(* Logix 5000 project; controller AMP_Servo_Demo vendor 1 type 14 code 154 rev 32.15; software revision 32.05; part 4 of 5 *)

ADD_ON_INSTRUCTION AMP_Relative_Move   (* revision 1.0, vendor Applied Motion Products Inc. *)
// Applied Motion - Motor Relative Move - AOI
// Help:
// The Relative Move AOI is used to move an axis by a specified distance (positive or negative) relative to its currently commanded position(FL).
VAR_IN_OUT
   Input : DINT[20]; {required}   // Drive Input Assembly
        [12]   // Digital_Outputs
        [7]   // Drive_Temperature
        [2]   // Control_Mode
        [3]   // Status_Code
        [9]   // Second_Encoder_Position
        [16]   // Analog_Input1
        [17]   // Analog_Input2
        [4]   // Alarm_Code
        [18]   // Torque_Limit
        [5]   // Supply_Voltage
        [6]   // Applied_Torque
        [10]   // Position_Error
        [13]   // Digital_Inputs
        [14]   // Analog_Output1
        [15]   // Analog_Output2
        [1]   // OpCode1_Received
        [8]   // Encoder_Position
        [0]   // Control_Word_Received
        [11]   // Actual_Velocity_RPS
        [19]   // Second_Encoder_Speed
   Output : DINT[11]; {required}   // Drive Output Assembly
        [0]   // Control Word
        [5]   // Porifle Acceleration
        [6]   // Profile Deceleration
        [7]   // Target Torque
        [4]   // Target Velocity
        [10]   // Reserved
        [3]   // Target Pos
        [1]   // OpCode 1
        [2]   // OpCode 2
        [8]   // OpCode 3
        [9]   // OpCode 4
END_VAR
VAR_INPUT
   Start : BOOL; {required}   // Start the Relative Move
   Distance : DINT; {required}   // Relative Distance to Move (negative = reverse)
   Speed_rps : REAL; {required}   // Velocity of Move (rev/sec)
   Acc : REAL; {required}   // Acceleration of Move (rev/s/s)
   Dec : REAL; {required}   // Deceleration of Move (rev/s/s)
END_VAR
VAR_OUTPUT
   Sent : BOOL; {access Read Only, visible}   // Move has been sent to drive
   In_Progress : BOOL; {access Read Only, visible}   // Move in progress
   Done : BOOL; {access Read Only, visible}   // Move completed without errors - desired position reached
   Error : BOOL; {access Read Only, visible}   // Move failed to complete - drive not ready or faulted
   State : DINT := 10; {access Read Only}   // Internal state of progress
END_VAR
VAR
   Loc_StatusCode : AMP_Status_Word_Servo; {access None}
   Loc_Rel_ONS : BOOL;
   Loc_Input_Assembly : AMP_Input_Assembly_Servo_v2; {access None}
   Loc_Command_Timeout : TIMER := (PRE := 2000); {access None}   // Timer to output fault if command is not Done
END_VAR

ROUTINE Logic   (* ladder *)
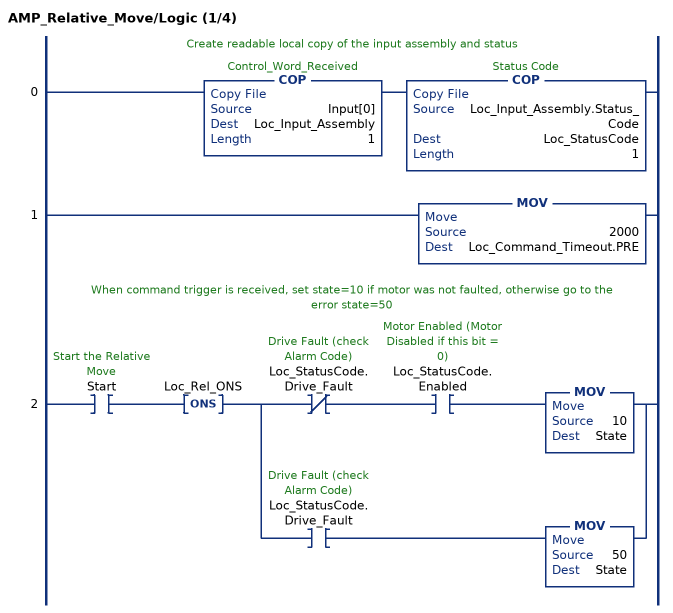
   // Create readable local copy of the input assembly and status
   0: COP(Input[0],Loc_Input_Assembly,1)COP(Loc_Input_Assembly.Status_Code,Loc_StatusCode,1);
   1: MOV(2000,Loc_Command_Timeout.PRE);
   // When command trigger is received, set state=10 if motor was not faulted, otherwise go to the error state=50
   2: XIC(Start)ONS(Loc_Rel_ONS)[XIO(Loc_StatusCode.Drive_Fault) XIC(Loc_StatusCode.Enabled) MOV(10,State) ,XIC(Loc_StatusCode.Drive_Fault) MOV(50,State) ];
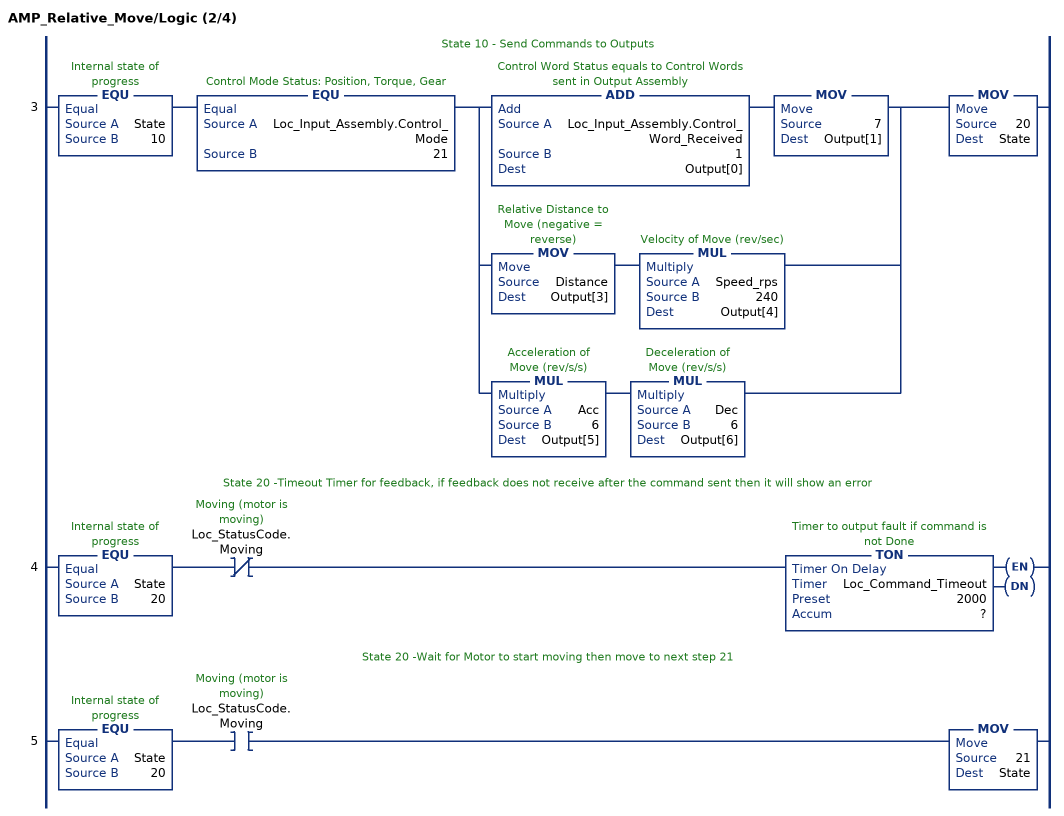
   // State 10 - Send Commands to Outputs
   3: EQU(State,10)EQU(Loc_Input_Assembly.Control_Mode,21)[ADD(Loc_Input_Assembly.Control_Word_Received,1,Output[0]) MOV(7,Output[1]) ,MOV(Distance,Output[3]) MUL(Speed_rps,240,Output[4]) ,MUL(Acc,6,Output[5]) MUL(Dec,6,Output[6]) ]MOV(20,State);
   // State 20 -Timeout Timer for feedback, if feedback does not receive after the command sent then it will show an error
   4: EQU(State,20)XIO(Loc_StatusCode.Moving)TON(Loc_Command_Timeout,?,?);
   // State 20 -Wait for Motor to start moving then move to next step 21
   5: EQU(State,20)XIC(Loc_StatusCode.Moving)MOV(21,State);
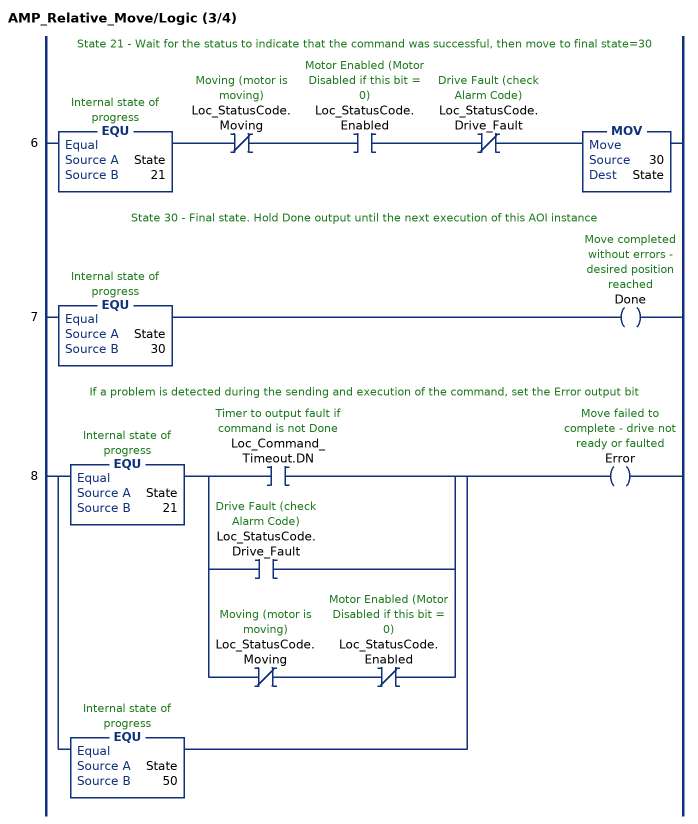
   // State 21 - Wait for the status to indicate that the command was successful, then move to final state=30
   6: EQU(State,21)XIO(Loc_StatusCode.Moving)XIC(Loc_StatusCode.Enabled)XIO(Loc_StatusCode.Drive_Fault)MOV(30,State);
   // State 30 - Final state. Hold Done output until the next execution of this AOI instance
   7: EQU(State,30)OTE(Done);
   // If a problem is detected during the sending and execution of the command, set the Error output bit
   8: [EQU(State,21) [XIC(Loc_Command_Timeout.DN) ,XIC(Loc_StatusCode.Drive_Fault) ,XIO(Loc_StatusCode.Moving) XIO(Loc_StatusCode.Enabled) ] ,EQU(State,50) ]OTE(Error);
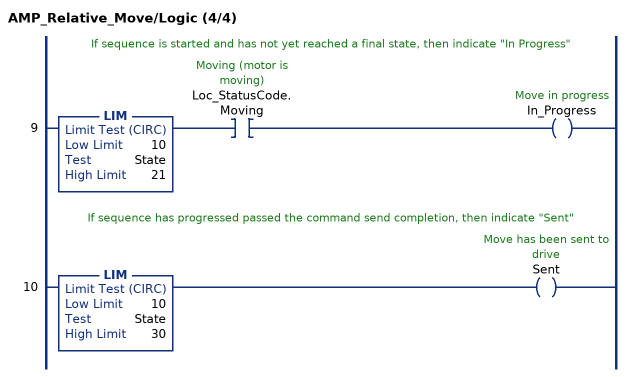
   // If sequence is started and has not yet reached a final state, then indicate "In Progress"
   9: LIM(10,State,21)XIC(Loc_StatusCode.Moving)OTE(In_Progress);
   // If sequence has progressed passed the command send completion, then indicate "Sent"
   10: LIM(10,State,30)OTE(Sent);
END_ROUTINE
END_ADD_ON_INSTRUCTION

ADD_ON_INSTRUCTION AMP_SCL_Command   (* revision 1.0, vendor Applied Motion Products Inc. *)
// Applied Motion - Motor SCL Command - AOI
// Help:
// The SCL Command Execute AOI executes selected SCL commands (as listed under “Available SCL Commands” in the reference manual).
VAR_IN_OUT
   Input : DINT[20]; {required}   // Drive Input Assembly
        [12]   // Digital_Outputs
        [7]   // Drive_Temperature
        [2]   // Control_Mode
        [9]   // Second_Encoder_Position
        [3]   // Status_Code
        [16]   // Analog_Input1
        [17]   // Analog_Input2
        [18]   // Torque_Limit
        [4]   // Alarm_Code
        [5]   // Supply_Voltage
        [6]   // Applied_Torque
        [10]   // Position_Error
        [13]   // Digital_Inputs
        [14]   // Analog_Output1
        [15]   // Analog_Output2
        [1]   // OpCode1_Received
        [8]   // Encoder_Position
        [0]   // Control_Word_Received
        [11]   // Actual_Velocity_RPS
        [19]   // Second_Encoder_Speed
   Output : DINT[11]; {required}   // Drive Output Assembly
        [0]   // Control Word
        [5]   // Porifle Acceleration
        [6]   // Profile Deceleration
        [7]   // Target Torque
        [4]   // Target Velocity
        [10]   // Reserved
        [3]   // Target Pos
        [1]   // OpCode 1
        [2]   // OpCode 2
        [8]   // OpCode 3
        [9]   // OpCode 4
END_VAR
VAR_INPUT
   Execute : BOOL; {required}   // Execute the SCL command
   SCL_Command : INT; {required}   // SCL Command Characters (always 2)
   Reg1 : DINT; {required}   // Data / SCL Register 1
   Reg2 : DINT; {required}   // Data / SCL Register 2
END_VAR
VAR_OUTPUT
   Sent : BOOL; {access Read Only, visible}   // Command has been sent to drive
   In_Progress : BOOL; {access Read Only, visible}   // Command in progress
   Done : BOOL; {access Read Only, visible}   // Command completed without errors
   Error : BOOL; {access Read Only, visible}   // Command failed
   State : DINT := 10; {access Read Only}   // Internal state of progress
END_VAR
VAR
   Loc_StatusCode : AMP_Status_Word_Servo; {access None}
   Loc_SCL_ONS : BOOL;
   Loc_Input_Assembly : AMP_Input_Assembly_Servo_v2; {access None}
END_VAR

ROUTINE Logic   (* ladder *)
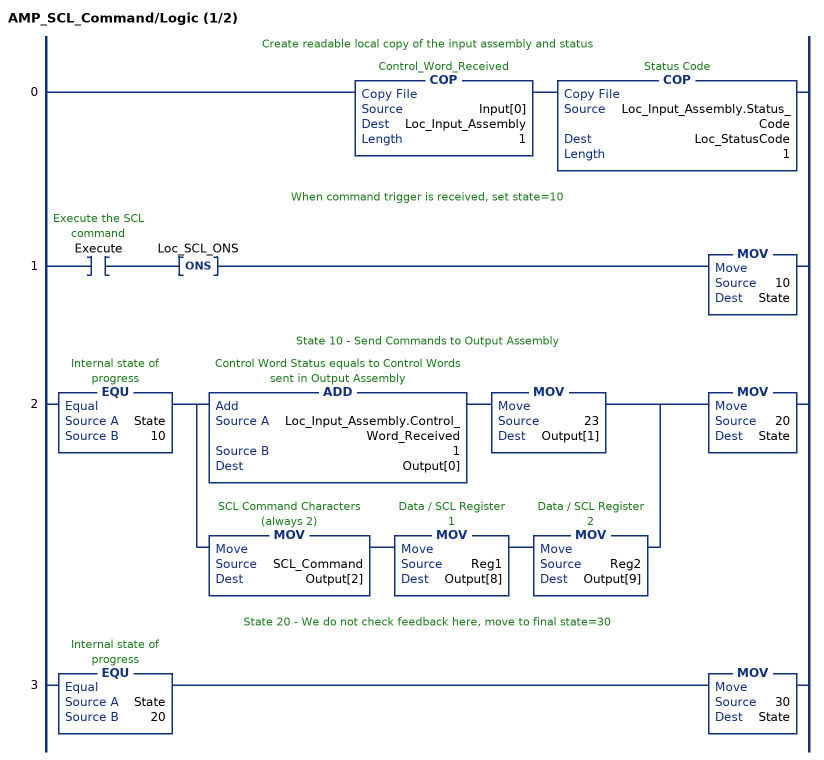
   // Create readable local copy of the input assembly and status
   0: COP(Input[0],Loc_Input_Assembly,1)COP(Loc_Input_Assembly.Status_Code,Loc_StatusCode,1);
   // When command trigger is received, set state=10
   1: XIC(Execute)ONS(Loc_SCL_ONS)MOV(10,State);
   // State 10 - Send Commands to Output Assembly
   2: EQU(State,10)[ADD(Loc_Input_Assembly.Control_Word_Received,1,Output[0]) MOV(23,Output[1]) ,MOV(SCL_Command,Output[2]) MOV(Reg1,Output[8]) MOV(Reg2,Output[9]) ]MOV(20,State);
   // State 20 - We do not check feedback here, move to final state=30
   3: EQU(State,20)MOV(30,State);
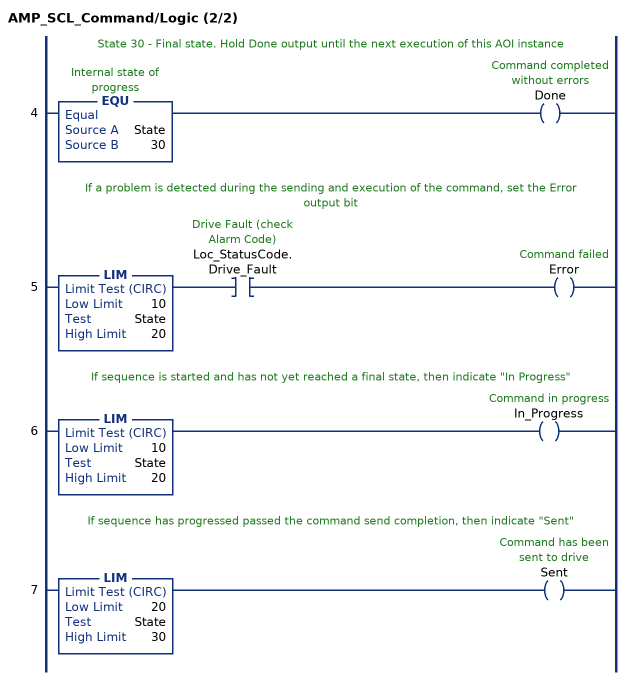
   // State 30 - Final state. Hold Done output until the next execution of this AOI instance
   4: EQU(State,30)OTE(Done);
   // If a problem is detected during the sending and execution of the command, set the Error output bit
   5: LIM(10,State,20)XIC(Loc_StatusCode.Drive_Fault)OTE(Error);
   // If sequence is started and has not yet reached a final state, then indicate "In Progress"
   6: LIM(10,State,20)OTE(In_Progress);
   // If sequence has progressed passed the command send completion, then indicate "Sent"
   7: LIM(20,State,30)OTE(Sent);
END_ROUTINE
END_ADD_ON_INSTRUCTION

ADD_ON_INSTRUCTION AMP_Set_Position   (* revision 1.0 *)
// Applied Motion - Motor Set Position - AOI
// Help:
// The Motor Enable AOI restores drive current to motor.
VAR_IN_OUT
   Input : DINT[20]; {required}   // Drive Input Assembly
        [12]   // Digital_Outputs
        [7]   // Drive_Temperature
        [2]   // Control_Mode
        [3]   // Status_Code
        [9]   // Second_Encoder_Position
        [16]   // Analog_Input1
        [17]   // Analog_Input2
        [4]   // Alarm_Code
        [18]   // Torque_Limit
        [5]   // Supply_Voltage
        [6]   // Applied_Torque
        [10]   // Position_Error
        [13]   // Digital_Inputs
        [14]   // Analog_Output1
        [15]   // Analog_Output2
        [1]   // OpCode1_Received
        [0]   // Control_Word_Received
        [11]   // Actual_Velocity_RPS
        [8]   // Encoder_Position
        [19]   // Second_Encoder_Speed
   Output : DINT[11]; {required}   // Drive Output Assembly
        [0]   // Control Word
        [5]   // Porifle Acceleration
        [6]   // Profile Deceleration
        [7]   // Target Torque
        [4]   // Target Velocity
        [10]   // Reserved
        [3]   // Target Pos
        [1]   // OpCode 1
        [2]   // OpCode 2
        [8]   // OpCode 3
        [9]   // OpCode 4
END_VAR
VAR_INPUT
   Execute : BOOL; {required}   // Execute the SCL command EP
   Position : DINT; {required}   // Position SetPoint DINT value
END_VAR
VAR_OUTPUT
   Sent : BOOL; {access Read Only, visible}   // Command has been sent to drive
   In_Progress : BOOL; {access Read Only, visible}   // Command in progress
   Done : BOOL; {access Read Only, visible}   // Command completed without errors - Drive is Homed
   Error : BOOL; {access Read Only, visible}   // Command failed
   State : DINT := 10; {access Read Only}   // Internal state of progress
END_VAR
VAR
   Loc_StatusCode : AMP_Status_Word_Servo;
   Loc_Input_Assembly : AMP_Input_Assembly_Servo_v2;
   Loc_SCL_ONS : BOOL;
   Loc_Reg2 : DINT;   // Data / SCL Register 2
   Loc_Reg1 : DINT;   // Data / SCL Register 1
   Loc_SCL_Command : INT := 'EP';   // SCL Command Characters (always 2)
END_VAR

ROUTINE Logic   (* ladder *)
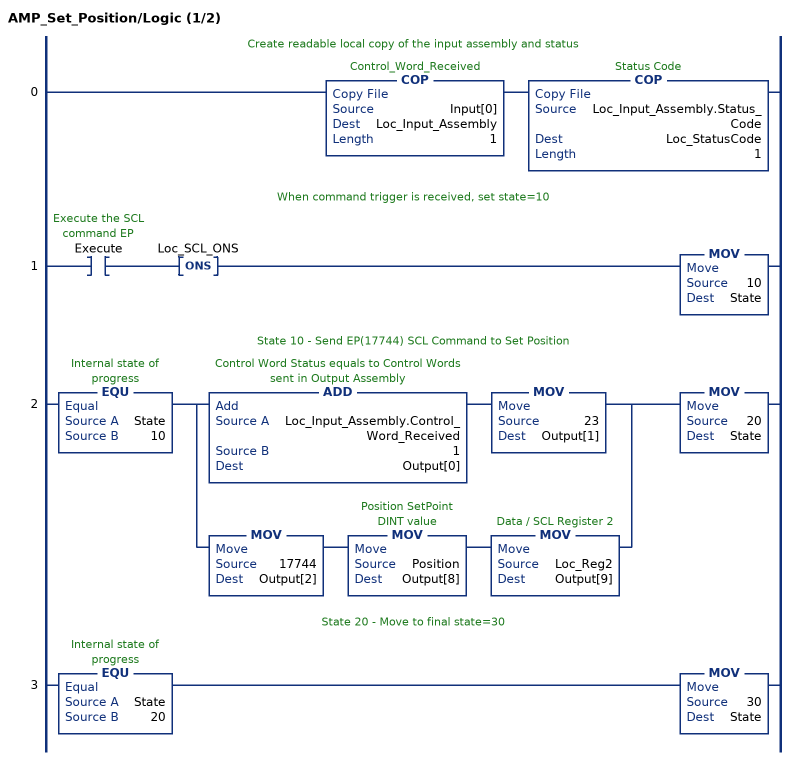
   // Create readable local copy of the input assembly and status
   0: COP(Input[0],Loc_Input_Assembly,1)COP(Loc_Input_Assembly.Status_Code,Loc_StatusCode,1);
   // When command trigger is received, set state=10
   1: XIC(Execute)ONS(Loc_SCL_ONS)MOV(10,State);
   // State 10 - Send EP(17744) SCL Command to Set Position
   2: EQU(State,10)[ADD(Loc_Input_Assembly.Control_Word_Received,1,Output[0]) MOV(23,Output[1]) ,MOV(17744,Output[2]) MOV(Position,Output[8]) MOV(Loc_Reg2,Output[9]) ]MOV(20,State);
   // State 20 - Move to final state=30
   3: EQU(State,20)MOV(30,State);
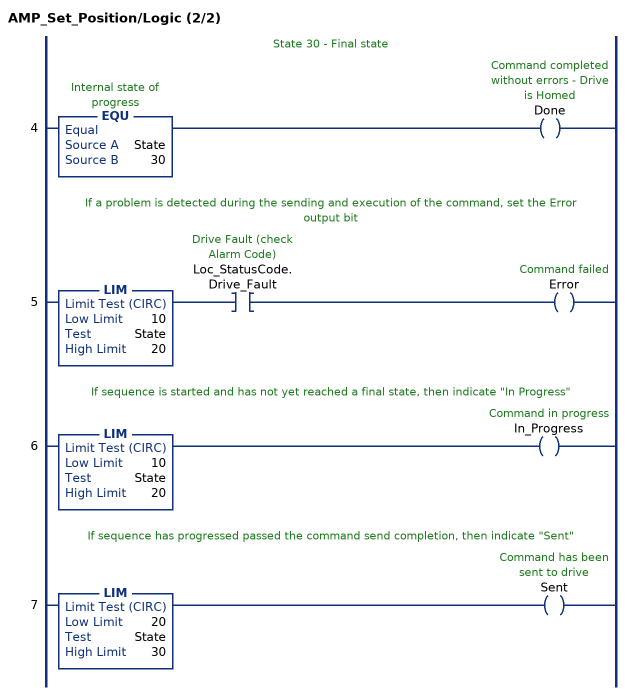
   // State 30 - Final state
   4: EQU(State,30)OTE(Done);
   // If a problem is detected during the sending and execution of the command, set the Error output bit
   5: LIM(10,State,20)XIC(Loc_StatusCode.Drive_Fault)OTE(Error);
   // If sequence is started and has not yet reached a final state, then indicate "In Progress"
   6: LIM(10,State,20)OTE(In_Progress);
   // If sequence has progressed passed the command send completion, then indicate "Sent"
   7: LIM(20,State,30)OTE(Sent);
END_ROUTINE
END_ADD_ON_INSTRUCTION

ADD_ON_INSTRUCTION AMP_Status_Code   (* revision 1.0, vendor Applied Motion Products Inc. *)
// Applied Motion - Status Code(SC) AOI
// Help:
// The Status Code AOI uses the raw data stored in the Status Code word (Element 0 from Input Assembly) to set individual appropriately named boolean outputs.
VAR_INPUT
   Input : DINT; {required}   // Element 4 from Drive Input Assembly
END_VAR
VAR_OUTPUT
   Motor_Enabled : BOOL; {access Read Only, visible}   // Motor is Enabled(Brake is released if applicable)
   Sampling : BOOL; {access Read Only, visible}   // Sampling (Luna software oscilloscope function opens)
   Drive_Fault : BOOL; {access Read Only, visible}   // Drive has fault, Motor Disabled
   In_Position : BOOL; {access Read Only, visible}   // Motor is in Position, it is standstill
   Moving : BOOL; {access Read Only, visible}   // Motor is Moving
   Jogging : BOOL; {access Read Only, visible}   // Motor is Jogging
   Stopping : BOOL; {access Read Only, visible}   // Motor is Stopping (Decelerating)
   Waiting : BOOL; {access Read Only, visible}   // Wait for Input Signal (e.g. follow WI command)
   Saving : BOOL; {access Read Only, visible}   // Drive is Saving Parameters
   Alarm_Present : BOOL; {access Read Only, visible}   // Dirve has alram present, fault and warning
   Homing : BOOL; {access Read Only, visible}   // Motor is Homing
   Wait_Time : BOOL; {access Read Only, visible}   // Waiting for an input (executing WD or WT command/delay after homing)
   Wizard_Running : BOOL; {access Read Only, visible}   // Wizard Running, Drive internal status
   Checking_Encoder : BOOL; {access Read Only, visible}   // Drive is checking encoder, Drive internal status
   Q_Program_Running : BOOL; {access Read Only, visible}   // Q Program is executing
   Servo_Ready : BOOL; {access Read Only, visible}   // Servo is ready
   CSP_Following : BOOL; {access Read Only, visible}   // CSP following internal status
   In_Velocity : BOOL; {access Read Only, visible}   // Motor is in Velocity
   Zero_Speed : BOOL; {access Read Only, visible}   // Motor is not moving
   Torque_Reached : BOOL; {access Read Only, visible}   // Torque Arrival
   In_Torque : BOOL; {access Read Only, visible}   // Consistent Torque
   Group2_PID : BOOL; {access Read Only, visible}   // The second set of gain is in operation
   Secondary_Control_Mode : BOOL; {access Read Only, visible}   // The second control mode is in operation
   Velocity_Reached : BOOL; {access Read Only, visible}   // Velocity is reached
   Homing_Complete : BOOL; {access Read Only, visible}   // Homing has been completed
END_VAR

ROUTINE Logic   (* ladder *)
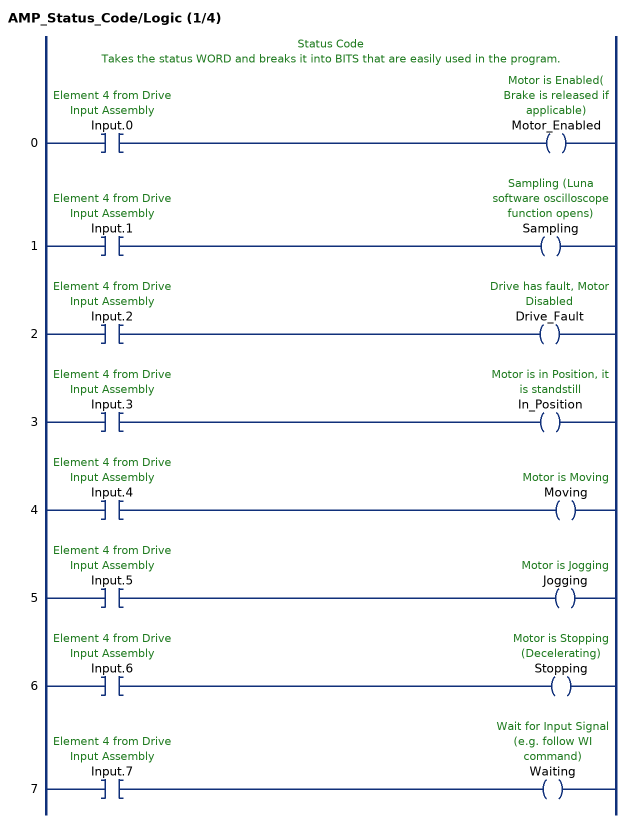
   // Status Code
   // Takes the status WORD and breaks it into BITS that are easily used in the program.
   0: XIC(Input.0)OTE(Motor_Enabled);
   1: XIC(Input.1)OTE(Sampling);
   2: XIC(Input.2)OTE(Drive_Fault);
   3: XIC(Input.3)OTE(In_Position);
   4: XIC(Input.4)OTE(Moving);
   5: XIC(Input.5)OTE(Jogging);
   6: XIC(Input.6)OTE(Stopping);
   7: XIC(Input.7)OTE(Waiting);
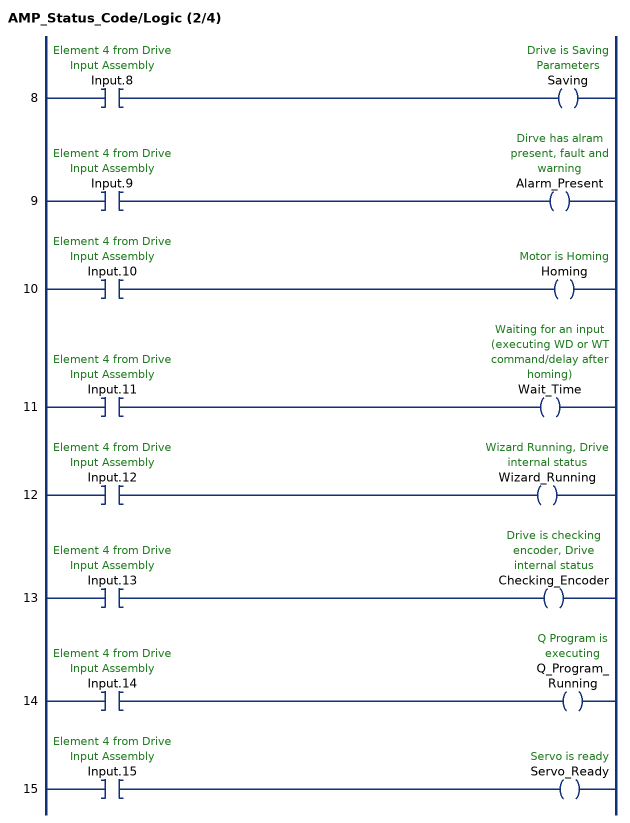
   8: XIC(Input.8)OTE(Saving);
   9: XIC(Input.9)OTE(Alarm_Present);
   10: XIC(Input.10)OTE(Homing);
   11: XIC(Input.11)OTE(Wait_Time);
   12: XIC(Input.12)OTE(Wizard_Running);
   13: XIC(Input.13)OTE(Checking_Encoder);
   14: XIC(Input.14)OTE(Q_Program_Running);
   15: XIC(Input.15)OTE(Servo_Ready);
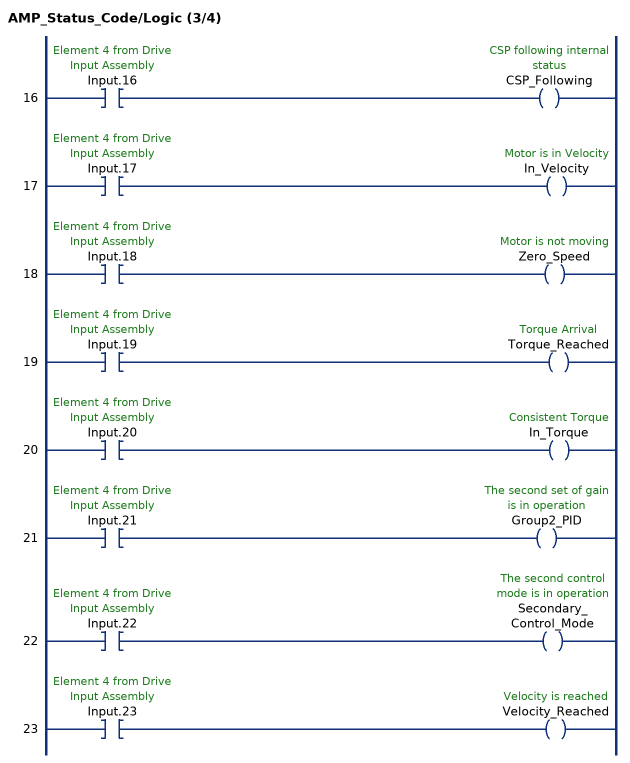
   16: XIC(Input.16)OTE(CSP_Following);
   17: XIC(Input.17)OTE(In_Velocity);
   18: XIC(Input.18)OTE(Zero_Speed);
   19: XIC(Input.19)OTE(Torque_Reached);
   20: XIC(Input.20)OTE(In_Torque);
   21: XIC(Input.21)OTE(Group2_PID);
   22: XIC(Input.22)OTE(Secondary_Control_Mode);
   23: XIC(Input.23)OTE(Velocity_Reached);
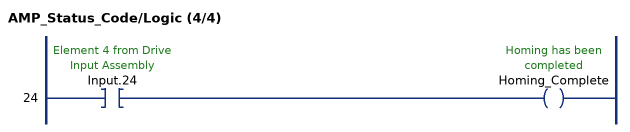
   24: XIC(Input.24)OTE(Homing_Complete);
END_ROUTINE
END_ADD_ON_INSTRUCTION

ADD_ON_INSTRUCTION AMP_Torque_Control   (* revision 1.0 *)
// Applied Motion - Motor Torque - AOI
// Use Normal/Crash Stop AOI to Stop Torque
// Help:
// The AOI switch Control mode to Torque mode and apply Torque. Use Normal stop or Crash stop AOI to stop applying torque.
// Target Torque Percentage is Limit by Torque Limit shown in Input Assembly.
VAR_IN_OUT
   Input : DINT[20]; {required}   // Drive Input Assembly
        [12]   // Digital_Outputs
        [7]   // Drive_Temperature
        [2]   // Control_Mode
        [3]   // Status_Code
        [16]   // Analog_Input1
        [17]   // Analog_Input2
        [9]   // Second_Encoder_Position
        [4]   // Alarm_Code
        [18]   // Torque_Limit
        [5]   // Supply_Voltage
        [6]   // Applied_Torque
        [0]   // Control_Word_Received
        [11]   // Actual_Velocity_RPS
        [19]   // Second_Encoder_Speed
        [10]   // Position_Error
        [13]   // Digital_Inputs
        [14]   // Analog_Output1
        [15]   // Analog_Output2
        [1]   // OpCode1_Received
        [8]   // Encoder_Position
   Output : DINT[11]; {required}   // Drive Output Assembly
        [0]   // Control Word
        [5]   // Porifle Acceleration
        [6]   // Profile Deceleration
        [7]   // Target Torque
        [4]   // Target Velocity
        [10]   // Reserved
        [3]   // Target Pos
        [1]   // OpCode 1
        [2]   // OpCode 2
        [8]   // OpCode 3
        [9]   // OpCode 4
END_VAR
VAR_INPUT
   Start : BOOL; {required}   // Start Applying Torque (on rising edge)
   Target_Torque_Percentage : INT := 10; {required}   // Target Torque Percentage, for reverse direction use Negative value
   Torque_Ramp : INT; {required}   // Torque Ramp (0.1%/sec)
   Speed_Limit_rps : REAL; {required}   // Torque Speed Limit in rps
   Acc : REAL; {required}   // Acceleration rev/s/s
   Dec : REAL; {required}   // Deceleration rev/s/s
END_VAR
VAR_OUTPUT
   Sent : BOOL; {access Read Only, visible}   // Command has been sent to drive
   In_Progress : BOOL; {access Read Only, visible}   // Command is in progress
   Done : BOOL; {access Read Only, visible}   // Command completed without errors
   Error : BOOL; {access Read Only, visible}   // Command Failed
   State : DINT := 10; {access Read Only}   // Internal state of progress
END_VAR
VAR
   Loc_StatusCode : AMP_Status_Word_Servo;
   Loc_Input_Assembly : AMP_Input_Assembly_Servo_v2;
   Loc_Torque_ONS : BOOL;
   Loc_Command_Wait : TIMER := (PRE := 100); {access None}   // Wait Timer for New Command
END_VAR

ROUTINE Logic   (* ladder *)
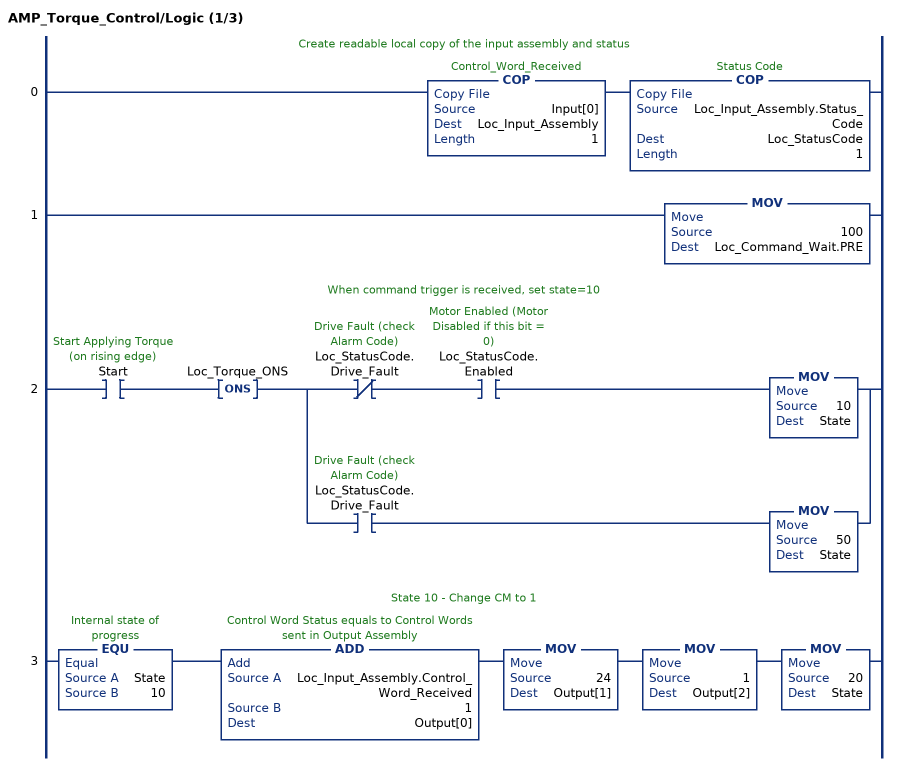
   // Create readable local copy of the input assembly and status
   0: COP(Input[0],Loc_Input_Assembly,1)COP(Loc_Input_Assembly.Status_Code,Loc_StatusCode,1);
   1: MOV(100,Loc_Command_Wait.PRE);
   // When command trigger is received, set state=10
   2: XIC(Start)ONS(Loc_Torque_ONS)[XIO(Loc_StatusCode.Drive_Fault) XIC(Loc_StatusCode.Enabled) MOV(10,State) ,XIC(Loc_StatusCode.Drive_Fault) MOV(50,State) ];
   // State 10 - Change CM to 1
   3: EQU(State,10)ADD(Loc_Input_Assembly.Control_Word_Received,1,Output[0])MOV(24,Output[1])MOV(1,Output[2])MOV(20,State);
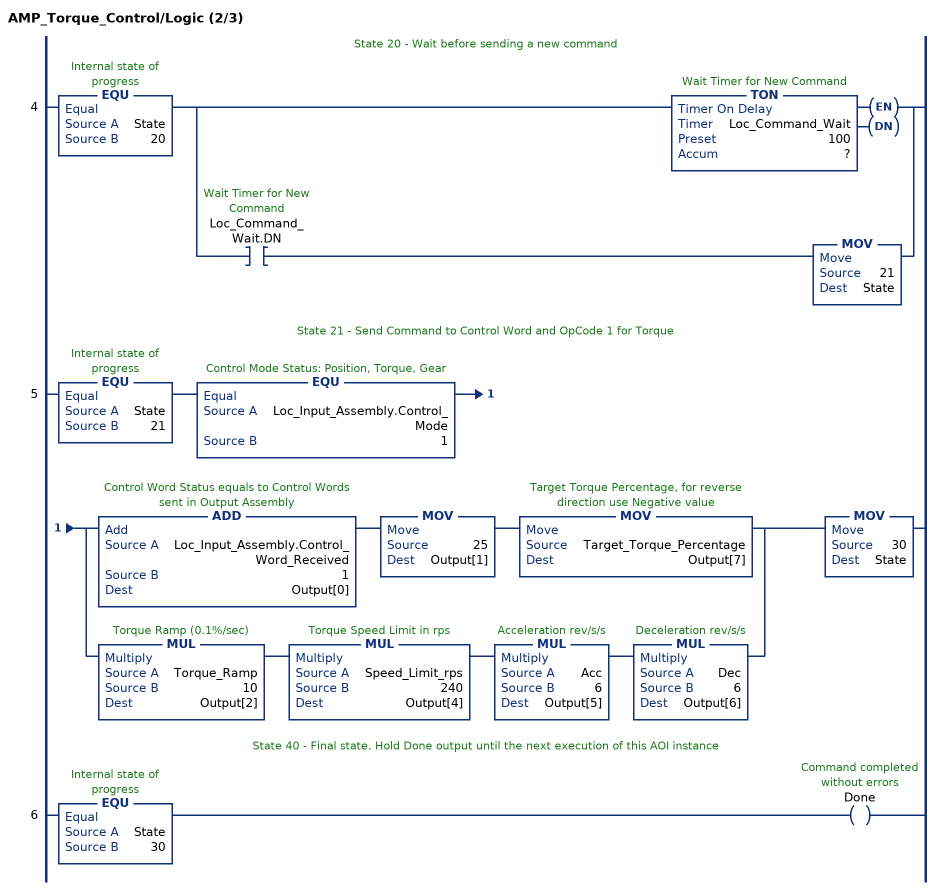
   // State 20 - Wait before sending a new command
   4: EQU(State,20)[TON(Loc_Command_Wait,?,?) ,XIC(Loc_Command_Wait.DN) MOV(21,State) ];
   // State 21 - Send Command to Control Word and OpCode 1 for Torque
   5: EQU(State,21)EQU(Loc_Input_Assembly.Control_Mode,1)[ADD(Loc_Input_Assembly.Control_Word_Received,1,Output[0]) MOV(25,Output[1]) MOV(Target_Torque_Percentage,Output[7]) ,MUL(Torque_Ramp,10,Output[2]) MUL(Speed_Limit_rps,240,Output[4]) MUL(Acc,6,Output[5]) MUL(Dec,6,Output[6]) ]MOV(30,State);
   // State 40 - Final state. Hold Done output until the next execution of this AOI instance
   6: EQU(State,30)OTE(Done);
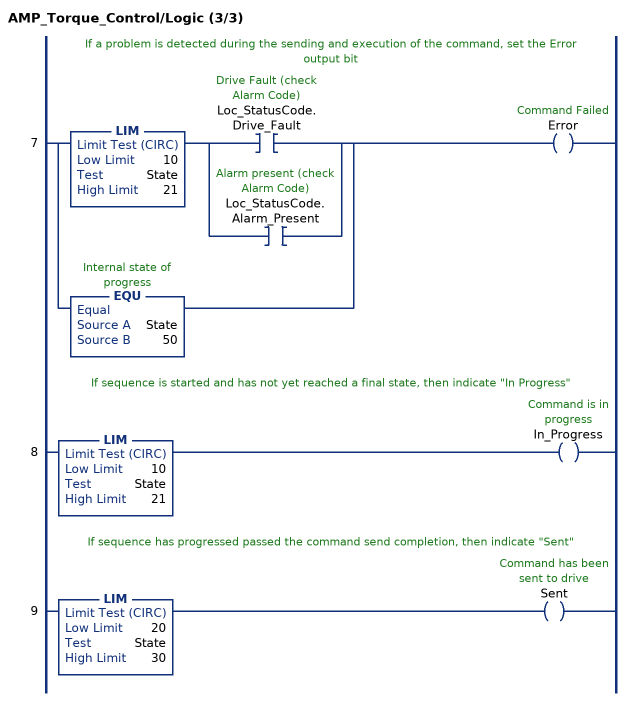
   // If a problem is detected during the sending and execution of the command, set the Error output bit
   7: [LIM(10,State,21) [XIC(Loc_StatusCode.Drive_Fault) ,XIC(Loc_StatusCode.Alarm_Present) ] ,EQU(State,50) ]OTE(Error);
   // If sequence is started and has not yet reached a final state, then indicate "In Progress"
   8: LIM(10,State,21)OTE(In_Progress);
   // If sequence has progressed passed the command send completion, then indicate "Sent"
   9: LIM(20,State,30)OTE(Sent);
END_ROUTINE
END_ADD_ON_INSTRUCTION

ADD_ON_INSTRUCTION AMP_Update_Jog_Speed   (* revision 1.0 *)
// Applied Motion - Motor Update Speed for Jog Only- AOI
// Help:
// This AOI updates the Jogging Speed either in Positive or Negative direction(CS). User need to use Normal Stop or Crash Stop AOI to Stop Jogging.
VAR_IN_OUT
   Input : DINT[20]; {required}   // Drive Input Assembly
        [12]   // Digital_Outputs
        [7]   // Drive_Temperature
        [2]   // Control_Mode
        [3]   // Status_Code
        [9]   // Second_Encoder_Position
        [16]   // Analog_Input1
        [17]   // Analog_Input2
        [4]   // Alarm_Code
        [19]   // Second_Encoder_Speed
        [18]   // Torque_Limit
        [5]   // Supply_Voltage
        [0]   // Control_Word_Received
        [6]   // Applied_Torque
        [11]   // Actual_Velocity_RPS
        [10]   // Position_Error
        [13]   // Digital_Inputs
        [14]   // Analog_Output1
        [15]   // Analog_Output2
        [1]   // OpCode1_Received
        [8]   // Encoder_Position
   Output : DINT[11]; {required}   // Drive Output Assembly
        [4]   // Jog Speed (0.25 rev/min)
        [0]   // Control Word
        [5]   // Porifle Acceleration
        [6]   // Profile Deceleration
        [7]   // Target Torque
        [10]   // Reserved
        [3]   // Target Pos
        [1]   // OpCode 1
        [2]   // OpCode 2
        [8]   // OpCode 3
        [9]   // OpCode 4
END_VAR
VAR_INPUT
   Update : BOOL; {required}   // Update Speed Command
   Speed_rps : REAL; {required}   // Velocity of Jog (rev/sec)(negative=reverse)
END_VAR
VAR_OUTPUT
   Sent : BOOL; {access Read Only, visible}   // Update Speed Command has been sent to drive
   In_Progress : BOOL; {access Read Only, visible}   // Update Speed Command in progress
   Done : BOOL; {access Read Only, visible}   // Update Speed command completed without errors
   Error : BOOL; {access Read Only, visible}   // Command failed
   State : DINT := 10; {access Read Only}   // Internal state of progress
END_VAR
VAR
   Loc_StatusCode : AMP_Status_Word_Servo;
   Command_Timeout : TIMER := (PRE := 2000);   // Timer to make sure command value was 0 before sending a new command
   Loc_Input_Assembly : AMP_Input_Assembly_Servo_v2;
   Loc_Jog_ONS : BOOL;
   Command_Reset : TIMER; {access None}   // Timer to make sure command value was 0 before sending a new command
END_VAR

ROUTINE Logic   (* ladder *)
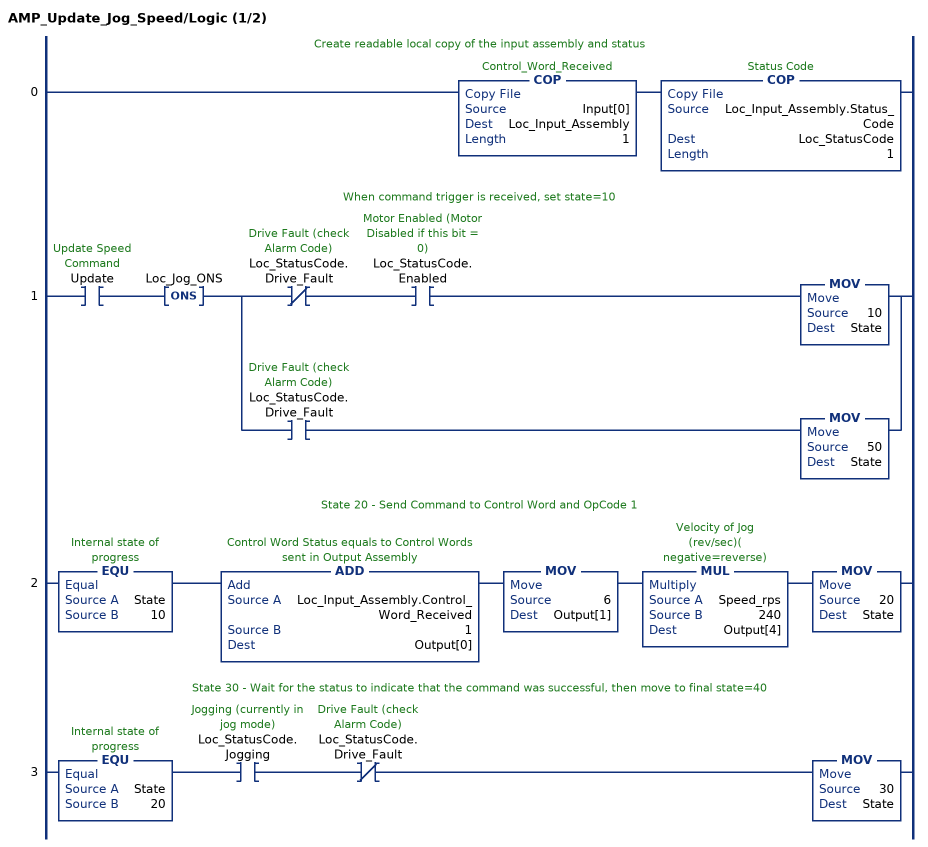
   // Create readable local copy of the input assembly and status
   0: COP(Input[0],Loc_Input_Assembly,1)COP(Loc_Input_Assembly.Status_Code,Loc_StatusCode,1);
   // When command trigger is received, set state=10
   1: XIC(Update)ONS(Loc_Jog_ONS)[XIO(Loc_StatusCode.Drive_Fault) XIC(Loc_StatusCode.Enabled) MOV(10,State) ,XIC(Loc_StatusCode.Drive_Fault) MOV(50,State) ];
   // State 20 - Send Command to Control Word and OpCode 1
   2: EQU(State,10)ADD(Loc_Input_Assembly.Control_Word_Received,1,Output[0])MOV(6,Output[1])MUL(Speed_rps,240,Output[4])MOV(20,State);
   // State 30 - Wait for the status to indicate that the command was successful, then move to final state=40
   3: EQU(State,20)XIC(Loc_StatusCode.Jogging)XIO(Loc_StatusCode.Drive_Fault)MOV(30,State);
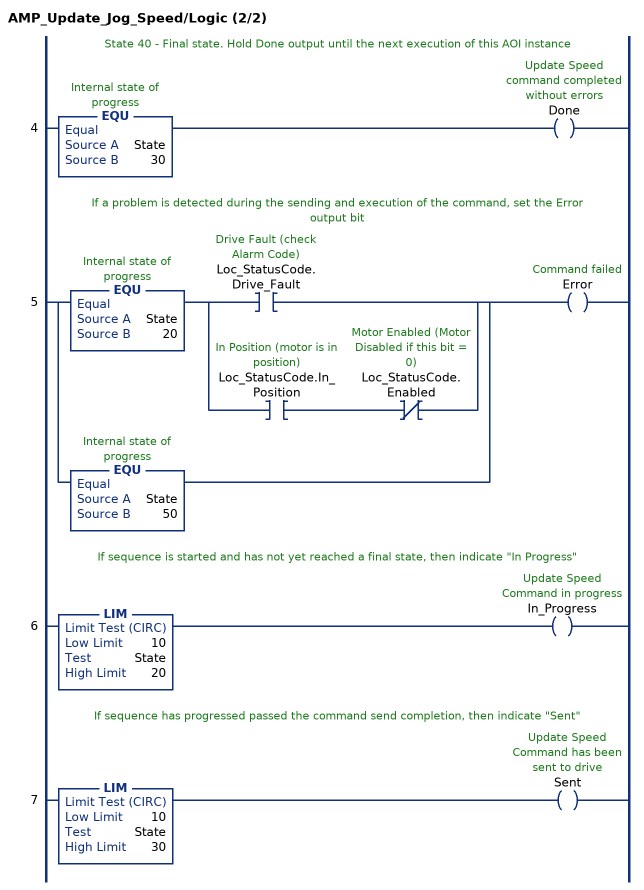
   // State 40 - Final state. Hold Done output until the next execution of this AOI instance
   4: EQU(State,30)OTE(Done);
   // If a problem is detected during the sending and execution of the command, set the Error output bit
   5: [EQU(State,20) [XIC(Loc_StatusCode.Drive_Fault) ,XIC(Loc_StatusCode.In_Position) XIO(Loc_StatusCode.Enabled) ] ,EQU(State,50) ]OTE(Error);
   // If sequence is started and has not yet reached a final state, then indicate "In Progress"
   6: LIM(10,State,20)OTE(In_Progress);
   // If sequence has progressed passed the command send completion, then indicate "Sent"
   7: LIM(10,State,30)OTE(Sent);
END_ROUTINE
END_ADD_ON_INSTRUCTION

VAR_GLOBAL   (* controller tags *)
   Amp_01_MSG1 : MESSAGE;
        MessageParameters(ServiceCode := 16#003c, LocalElement := Amp_01_MSG1_Param_Write[0], DestinationTag := Amp_01_MSG1_ReadParam_Response[0], ...)
   Amp_01_MSG1_Param_Req : SINT[8] := ([1] := 16#01, [3] := 16#9f);
        [7]   // Parameter (bit 0-7)
        [6]   // Parameter (bit 8-15)
        [2]   // Opcode (MSB)
        [3]   // Opcode (LSB)
        [0]   // Register Code
        [4]   // Parameter (bit 24-31)
        [5]   // Parameter (bit 16-23)
        [1]   // Message Type 1
   Amp_01_MSG1_Param_Write : SINT[8] := ([1] := 16#01, [3] := 16#9f);
        [7]   // Parameter (bit 0-7)
        [6]   // Parameter (bit 8-15)
        [2]   // Opcode (MSB)
        [3]   // Opcode (LSB)
        [0]   // Register Code
        [4]   // Parameter (bit 24-31)
        [5]   // Parameter (bit 16-23)
        [1]   // Message Type 1
   Amp_01_MSG1_ReadParam_Res_Read : SINT[8] := ([0] := 16#88, [1] := 16#02, [5] := 16#06, [6] := 16#80, [7] := 16#09);
        [2]   // Opcode (MSB)
        [3]   // Opcode (LSB)
        [4]   // Status/Data (bit 24-31)
        [5]   // Status/Data (bit 16-23)
        [0]   // Register Code
        [6]   // Status/Data (bit 8-15)
        [7]   // Status/Data (bit 0-7)
        [1]   // Message Type 1
   Amp_01_MSG1_ReadParam_Response : SINT[8] := ([1] := 16#01, [3] := 16#9f, [5] := 16#06, [6] := 16#80, [7] := 16#09);
        [2]   // Opcode (MSB)
        [3]   // Opcode (LSB)
        [4]   // Status/Data (bit 24-31)
        [5]   // Status/Data (bit 16-23)
        [0]   // Register Code
        [6]   // Status/Data (bit 8-15)
        [7]   // Status/Data (bit 0-7)
        [1]   // Message Type 1
   Amp_01_MSG2 : MESSAGE;
        MessageParameters(ServiceCode := 16#003c, LocalElement := Amp_01_MSG2_Param_Write[0], DestinationTag := Amp_01_MSG2_ReadParam_Response[0], ...)
   Amp_01_MSG2_Param_Req : SINT[8] := ([0] := 16#88);
        [0]   // Opcode
        [7]   // Parameter (bit 0-7)
        [1]   // Message Type
        [6]   // Parameter (bit 8-15)
        [2]   // Operand (MSB)
        [3]   // Operand (LSB)
        [4]   // Parameter (bit 24-31)
        [5]   // Parameter (bit 16-23)
   Amp_01_MSG2_Param_Write : SINT[8] := ([0] := 16#88, [1] := 16#02);
        [7]   // Parameter (bit 0-7)
        [0]   // Opcode
        [1]   // Message Type
        [6]   // Parameter (bit 8-15)
        [2]   // Operand (MSB)
        [3]   // Operand (LSB)
        [4]   // Parameter (bit 24-31)
        [5]   // Parameter (bit 16-23)
   Amp_01_MSG2_ReadParam_Res_Read : SINT[8] := ([5] := 16#0c, [6] := 16#56, [7] := 16#f0);
        [0]   // Opcode
        [7]   // Parameter (bit 0-7)
        [1]   // Message Type
        [6]   // Parameter (bit 8-15)
        [2]   // Operand (MSB)
        [3]   // Operand (LSB)
        [4]   // Parameter (bit 24-31)
        [5]   // Parameter (bit 16-23)
   Amp_01_MSG2_ReadParam_Response : SINT[8] := ([0] := 16#88, [1] := 16#02, [5] := 16#0c, [6] := 16#56, [7] := 16#f0);
        [0]   // Opcode
        [1]   // Message Type
        [2]   // Operand (MSB)
        [3]   // Operand (LSB)
   AMP_Axis1_Absolute_Move_Inst : AMP_Absolute_Move := (Position := 5000, Speed_rps := 2.0, Acc := 10.0, Dec := 10.0, Sent := 1, Done := 1, State := 30);
   AMP_Axis1_Alarm_Code_Inst : AMP_Alarm_Code;
   AMP_Axis1_Alarm_Reset_Inst : AMP_Alarm_Reset := (Sent := 1, Done := 1, State := 30);
   AMP_Axis1_Crash_Stop_Inst : AMP_Crash_Stop := (Sent := 1, Done := 1, State := 40);
   AMP_Axis1_DI_Monitor_Inst : AMP_DI_Monitor := (DI_1 := 1, DI_2 := 1, DI_3 := 1, DI_4 := 1);
   AMP_Axis1_DO_Control_Inst : AMP_DO_Control := (Output_Number := 1, Condition := 'L', DO_1 := 1, DO_3 := 1, DO_4 := 1, DO_5 := 1, DO_6 := 1);
   AMP_Axis1_Homing_Inst : AMP_Home := (Homing_Method := -1, Home_Speed_rps := 3.0, Home_Speed2_rps := 1.0, Home_Acc := 1.0, Home_Dec := 1.0, Hard_Stop_Homing_Torque := 3, Sent := 1, Done := 1, State := 40);
   AMP_Axis1_Inputs : AMP_Input_Assembly_Servo_v2 := (Control_Word_Received := -2147483631, OpCode1_Received := 8, Status_Code := 425984, Supply_Voltage := 230, Drive_Temperature := 328, Digital_Outputs := 2, Digital_Inputs := 15, Analog_Input1 := -34, Torque_Limit := 300);
   AMP_Axis1_Motor_Disable_Inst : AMP_Motor_Disable := (Sent := 1, Done := 1, State := 30);
   AMP_Axis1_Motor_Enable_Inst : AMP_Motor_Enable := (Sent := 1, Done := 1, State := 30);
   AMP_Axis1_Motor_Jog_Inst : AMP_Jog_Move := (Jog_Speed_rps := 5.0, Jog_Acc := 10.0, Jog_Dec := 10.0, Sent := 1, Done := 1, State := 30);
   AMP_Axis1_Normal_Stop_Inst : AMP_Normal_Stop := (Sent := 1, Done := 1, State := 40);
   AMP_Axis1_Point_to_Poinr_IO_Exec : AMP_Point_to_Point_IO := (Command := 'FS', IO1_Number := 3, IO1_Condition := 'H', IO2_Condition := '0', Distance := 20000, Speed := 1.0, Acc := 10.0, Dec := 10.0, Change_Distance := 25000, Change_Speed := 7.0, Sent := 1, Done := 1, State := 40);
   AMP_Axis1_Point_to_Point_FC_Exec : AMP_Point_to_Point_FC := (Distance := 120000, Speed := 0.3, Acc := 10.0, Dec := 10.0, Change_Distance := 30000, Change_Speed := 1.0, Sent := 1, Done := 1, State := 40);
   AMP_Axis1_Q_Segment_Execute_Inst : AMP_Q_Segment_Execute := (Q_Segment := 1, Sent := 1, Done := 1, State := 20);
   AMP_Axis1_Relative_Move_Inst : AMP_Relative_Move := (Distance := 250000, Speed_rps := 3.5, Acc := 5.0, Dec := 5.0, Sent := 1, Done := 1, State := 30);
   AMP_Axis1_SCL_Inst : AMP_SCL_Command := (SCL_Command := 'CC', Reg1 := 200, Sent := 1, Done := 1, State := 30);
   AMP_Axis1_Set_Position_Inst : AMP_Set_Position := (Position := 10000, Sent := 1, Done := 1, State := 30);
   AMP_Axis1_Status_Code_Inst : AMP_Status_Code := (Input := 16#0006_8000, Servo_Ready := 1, In_Velocity := 1, Zero_Speed := 1);
   AMP_Axis1_Torque_Inst : AMP_Torque_Control := (Target_Torque_Percentage := 3, Torque_Ramp := 1, Speed_Limit_rps := 5.0, Acc := 2.0, Dec := 2.0, Sent := 1, Done := 1, State := 30);
   AMP_Axis1_Update_Jog_Speed_Inst : AMP_Update_Jog_Speed := (Speed_rps := 10.0, Sent := 1, Done := 1, State := 30);
   AMP_Axis2_Absolute_Move_Inst : AMP_Absolute_Move := (Speed_rps := 1.0, Acc := 1.0, Dec := 1.0, Sent := 1, State := 20);
   AMP_Axis2_Alarm_Code_Inst : AMP_Alarm_Code;
   AMP_Axis2_Alarm_Reset_Inst : AMP_Alarm_Reset := (Sent := 1, Done := 1, State := 30);
   AMP_Axis2_Crash_Stop_Inst : AMP_Crash_Stop := (Sent := 1, Done := 1, State := 40);
   AMP_Axis2_DI_Monitor_Inst : AMP_DI_Monitor := (DI_1 := 1, DI_2 := 1, DI_3 := 1, DI_4 := 1, DI_5 := 1, DI_6 := 1, DI_7 := 1, DI_8 := 1);
   AMP_Axis2_DO_Control_Inst : AMP_DO_Control := (Output_Number := 1, Condition := 'H', DO_5 := 1, DO_6 := 1);
   AMP_Axis2_Homing_Inst : AMP_Home := (Homing_Method := -4, Home_Speed_rps := 1.0, Home_Speed2_rps := 1.0, Home_Acc := 1.0, Home_Dec := 1.0, Hard_Stop_Homing_Torque := 20, Sent := 1, Done := 1, State := 40);
   AMP_Axis2_Inputs : AMP_Input_Assembly_Servo_v2 := (Control_Word_Received := 305, OpCode1_Received := 8, Control_Mode := 21, Status_Code := 425993, Supply_Voltage := 3310, Applied_Torque := -4, Drive_Temperature := 503, Second_Encoder_Position := -3494654, Digital_Outputs := 15, Digital_Inputs := 255, Analog_Input1 := -10, Analog_Input2 := 3, Torque_Limit := 342);
   AMP_Axis2_Motor_Disable_Inst : AMP_Motor_Disable := (Sent := 1, Done := 1, State := 30);
   AMP_Axis2_Motor_Enable_Inst : AMP_Motor_Enable := (Sent := 1, Done := 1, State := 30);
   AMP_Axis2_Motor_Jog_Inst : AMP_Jog_Move := (Jog_Speed_rps := 1.0, Jog_Acc := 1.0, Jog_Dec := 1.0, Error := 1, State := 40);
   AMP_Axis2_Normal_Stop_Inst : AMP_Normal_Stop := (Sent := 1, Done := 1, State := 40);
   AMP_Axis2_Point_to_Poinr_IO_Exec : AMP_Point_to_Point_IO := (Command := 'FO', IO1_Number := 1, IO1_Condition := 'H', IO2_Number := 4, IO2_Condition := 'H', Distance := -3000, Speed := 1.0, Acc := 1.0, Dec := 1.0, Change_Distance := 2500, Change_Speed := 7.0, Sent := 1, Done := 1, State := 40);
   AMP_Axis2_Point_to_Point_FC_Exec : AMP_Point_to_Point_FC := (Distance := 50000, Speed := 0.3, Acc := 10.0, Dec := 10.0, Change_Distance := 10000, Change_Speed := 1.0, Sent := 1, Done := 1, State := 40);
   AMP_Axis2_Q_Segment_Execute_Inst : AMP_Q_Segment_Execute := (Q_Segment := 1, Sent := 1, Done := 1, State := 20);
   AMP_Axis2_Relative_Move_Inst : AMP_Relative_Move := (Distance := 25000, Speed_rps := 1.0, Acc := 5.0, Dec := 5.0, Sent := 1, Done := 1, State := 30);
   AMP_Axis2_SCL_Inst : AMP_SCL_Command := (SCL_Command := 'SP', Reg1 := 100, Sent := 1, Done := 1, State := 30);
   AMP_Axis2_Set_Position_Inst : AMP_Set_Position := (Sent := 1, Done := 1, State := 30);
   AMP_Axis2_Status_Code_Inst : AMP_Status_Code := (Input := 16#0006_8009, Motor_Enabled := 1, In_Position := 1, Servo_Ready := 1, In_Velocity := 1, Zero_Speed := 1);
   AMP_Axis2_Update_Jog_Speed_Inst : AMP_Update_Jog_Speed := (Speed_rps := 1.0, Sent := 1, Done := 1, State := 30);
   AMP_Axis2Torque_Inst : AMP_Torque_Control := (Target_Torque_Percentage := 20, Torque_Ramp := 50, Speed_Limit_rps := 0.5, Acc := 1.0, Dec := 1.0, Sent := 1, Done := 1, State := 30);
   AMP_Input_Axis1_Inst : AMP_Input_Assembly := (Control_Word_Received := -2147483631, OpCode1_Received := 8, Status_Code := 16#0006_8000, DC_Bus_Voltage := 23.1, Drive_Temperature_C := 32.8, Actual_Velocity_rps := 0.004166667, Digital_Output_Status := 2, Digital_Input_Status := 15, Analog_Input_1 := -35, Torque_Limit := 300);
   AMP_Input_Axis2_Inst : AMP_Input_Assembly := (Control_Word_Received := 305, OpCode1_Received := 8, Control_Mode_Active := 21, Status_Code := 16#0006_8009, DC_Bus_Voltage := 331.0, Applied_Torque_Percentage := -4.0, Drive_Temperature_C := 50.3, Digital_Output_Status := 15, Digital_Input_Status := 255, Analog_Input_1 := -10, Analog_Input_2 := 3, Torque_Limit := 342, External_Encoder_Position := -3494654);
END_VAR

PROGRAM Explicit_Messages   (* main routine MainRoutine *)
VAR
   Amp_01_MSG2_ReadParam_Active : BOOL;
   Amp_01_MSG2_ReadParam_Done_ONS : BOOL;
   Amp_01_MSG_ReadParam_Active : BOOL;
   Amp_01_MSG_ReadParam_Done_ONS : BOOL;
END_VAR

ROUTINE AMP_Servo_Axis1_Explicit   (* ladder *)
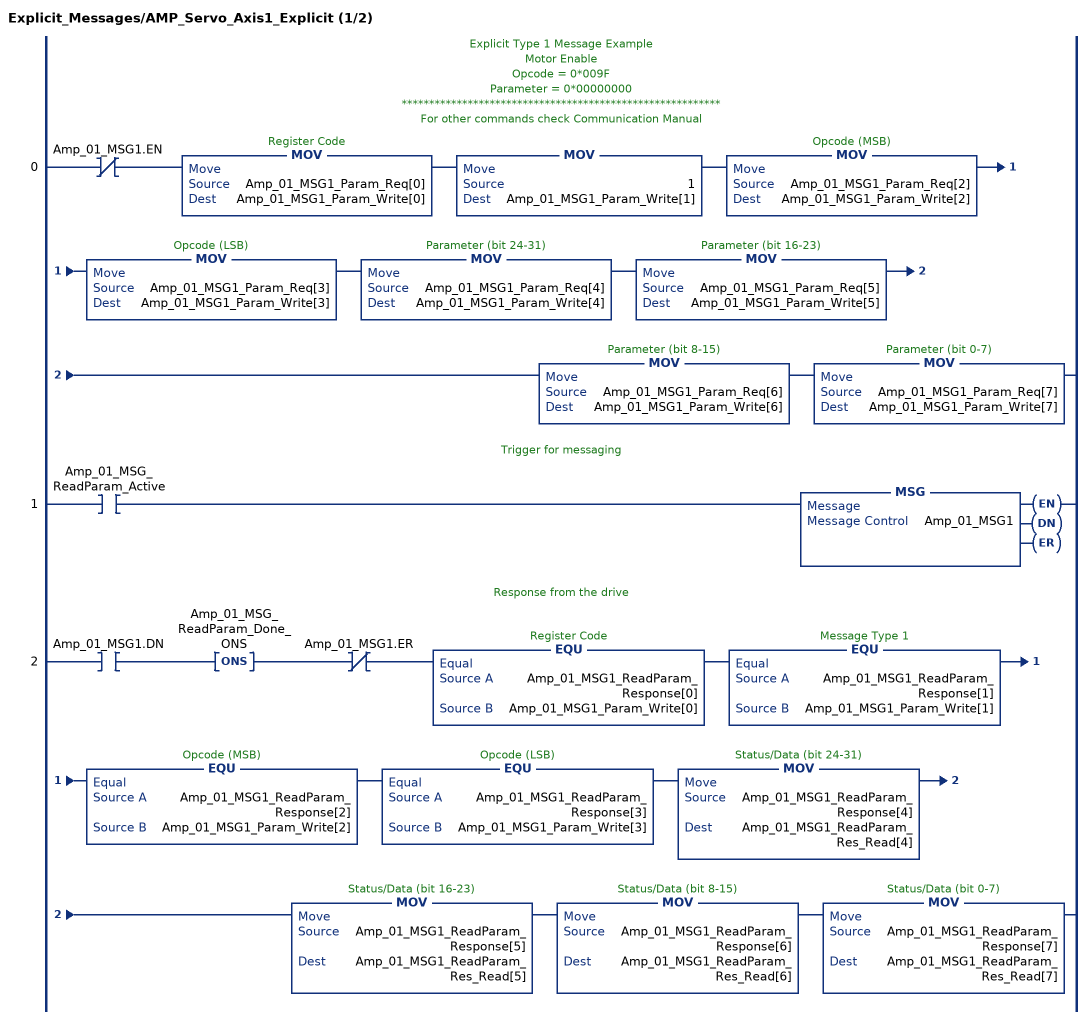
   // Explicit Type 1 Message Example
   // Motor Enable
   // Opcode = 0*009F
   // Parameter = 0*00000000
   // **********************************************************
   // For other commands check Communication Manual
   0: XIO(Amp_01_MSG1.EN)MOV(Amp_01_MSG1_Param_Req[0],Amp_01_MSG1_Param_Write[0])MOV(1,Amp_01_MSG1_Param_Write[1])MOV(Amp_01_MSG1_Param_Req[2],Amp_01_MSG1_Param_Write[2])MOV(Amp_01_MSG1_Param_Req[3],Amp_01_MSG1_Param_Write[3])MOV(Amp_01_MSG1_Param_Req[4],Amp_01_MSG1_Param_Write[4])MOV(Amp_01_MSG1_Param_Req[5],Amp_01_MSG1_Param_Write[5])MOV(Amp_01_MSG1_Param_Req[6],Amp_01_MSG1_Param_Write[6])MOV(Amp_01_MSG1_Param_Req[7],Amp_01_MSG1_Param_Write[7]);
   // Trigger for messaging
   1: XIC(Amp_01_MSG_ReadParam_Active)MSG(Amp_01_MSG1);
   // Response from the drive
   2: XIC(Amp_01_MSG1.DN)ONS(Amp_01_MSG_ReadParam_Done_ONS)XIO(Amp_01_MSG1.ER)EQU(Amp_01_MSG1_ReadParam_Response[0],Amp_01_MSG1_Param_Write[0])EQU(Amp_01_MSG1_ReadParam_Response[1],Amp_01_MSG1_Param_Write[1])EQU(Amp_01_MSG1_ReadParam_Response[2],Amp_01_MSG1_Param_Write[2])EQU(Amp_01_MSG1_ReadParam_Response[3],Amp_01_MSG1_Param_Write[3])MOV(Amp_01_MSG1_ReadParam_Response[4],Amp_01_MSG1_ReadParam_Res_Read[4])MOV(Amp_01_MSG1_ReadParam_Response[5],Amp_01_MSG1_ReadParam_Res_Read[5])MOV(Amp_01_MSG1_ReadParam_Response[6],Amp_01_MSG1_ReadParam_Res_Read[6])MOV(Amp_01_MSG1_ReadParam_Response[7],Amp_01_MSG1_ReadParam_Res_Read[7]);
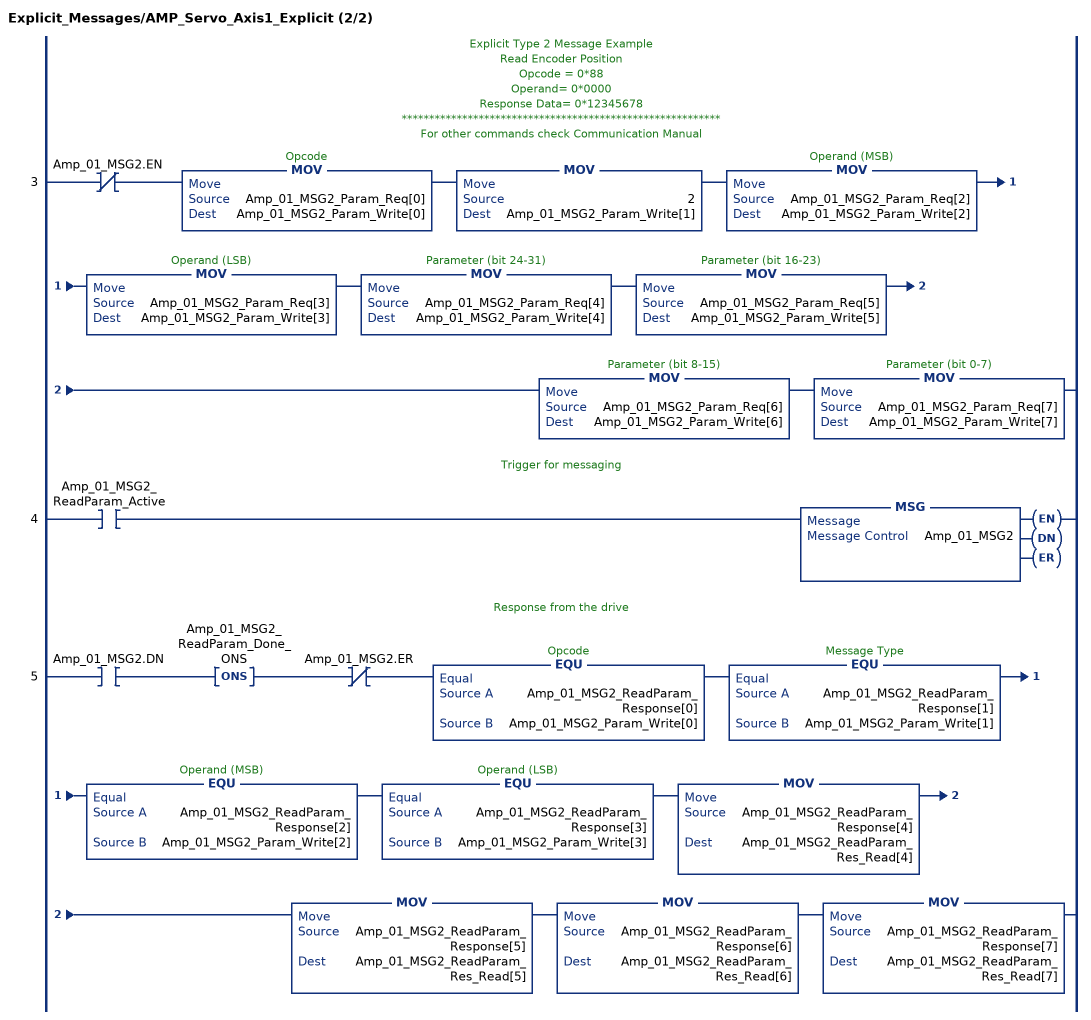
   // Explicit Type 2 Message Example
   // Read Encoder Position
   // Opcode = 0*88
   // Operand= 0*0000
   // Response Data= 0*12345678
   // **********************************************************
   // For other commands check Communication Manual
   3: XIO(Amp_01_MSG2.EN)MOV(Amp_01_MSG2_Param_Req[0],Amp_01_MSG2_Param_Write[0])MOV(2,Amp_01_MSG2_Param_Write[1])MOV(Amp_01_MSG2_Param_Req[2],Amp_01_MSG2_Param_Write[2])MOV(Amp_01_MSG2_Param_Req[3],Amp_01_MSG2_Param_Write[3])MOV(Amp_01_MSG2_Param_Req[4],Amp_01_MSG2_Param_Write[4])MOV(Amp_01_MSG2_Param_Req[5],Amp_01_MSG2_Param_Write[5])MOV(Amp_01_MSG2_Param_Req[6],Amp_01_MSG2_Param_Write[6])MOV(Amp_01_MSG2_Param_Req[7],Amp_01_MSG2_Param_Write[7]);
   // Trigger for messaging
   4: XIC(Amp_01_MSG2_ReadParam_Active)MSG(Amp_01_MSG2);
   // Response from the drive
   5: XIC(Amp_01_MSG2.DN)ONS(Amp_01_MSG2_ReadParam_Done_ONS)XIO(Amp_01_MSG2.ER)EQU(Amp_01_MSG2_ReadParam_Response[0],Amp_01_MSG2_Param_Write[0])EQU(Amp_01_MSG2_ReadParam_Response[1],Amp_01_MSG2_Param_Write[1])EQU(Amp_01_MSG2_ReadParam_Response[2],Amp_01_MSG2_Param_Write[2])EQU(Amp_01_MSG2_ReadParam_Response[3],Amp_01_MSG2_Param_Write[3])MOV(Amp_01_MSG2_ReadParam_Response[4],Amp_01_MSG2_ReadParam_Res_Read[4])MOV(Amp_01_MSG2_ReadParam_Response[5],Amp_01_MSG2_ReadParam_Res_Read[5])MOV(Amp_01_MSG2_ReadParam_Response[6],Amp_01_MSG2_ReadParam_Res_Read[6])MOV(Amp_01_MSG2_ReadParam_Response[7],Amp_01_MSG2_ReadParam_Res_Read[7]);
END_ROUTINE
